{attribute 'Tc2GvlVarNames' := ''}
VAR_GLOBAL
	MATH: exCONSTANTS_MATH;
	PHYS: exCONSTANTS_PHYS;

END_VAR

(* stored: Version 1.1.0.1, ProductVersion 3.1.4024.3
   GVL exGlobale_Variablen: Id {d4bcba04-5dbe-4420-a32d-15b51a8dd874} *)
